
FUNCTION CB_sub_tod_tod : TIME


TITLE = ' substracting two time of day '
VERSION : '1.0'
AUTHOR  : CB
NAME    : suTodTod
FAMILY  : TNI

VAR_INPUT
    IN0 : TOD ;
    IN1 : TOD ;
END_VAR

BEGIN
    CB_sub_tod_tod := IN0 - IN1;
END_FUNCTION
